// TwinCAT 3 PLC project PD30CTBxx
// Title: PD30CTBxx
// Company: iMusic AS
// Author: Jakob Bak
// ProjectVersion: 0.0.1.0
// Description: TwinCAT Library for PD30CTB* series Diffuse-reflective Photoelectric Sensors from Carlo Gavazzi
// ProgramVersion: 3.1.4024.0
// libraries:
//   Tc2_Standard, * (Beckhoff Automation GmbH)
//   Tc2_System, * (Beckhoff Automation GmbH)
//   Tc3_Module, * (Beckhoff Automation GmbH)
// project tree:
//   DUTs/ ST_PD30CTBxx.TcDUT
//   / PlcTask.TcTTO
//   POUs/ MAIN.TcPOU
//   Version/ Global_Version.TcGVL
// real-time tasks:
//   TASK PlcTask: cycle T#10ms, priority 20, ADS port 350

CONFIGURATION PD30CTBxx
    RESOURCE PLC ON TwinCAT3
        TASK PlcTask(INTERVAL := T#10ms, PRIORITY := 20);
        PROGRAM MAIN WITH PlcTask : MAIN;
    END_RESOURCE
END_CONFIGURATION

// ---- DUTs/ST_PD30CTBxx.TcDUT

TYPE ST_PD30CTBxx :
STRUCT
	bAnalogueValue				AT%I* : UINT;
	bSwitchingSignalChannel_1	AT%I* : BIT;
	bSwitchingSignalChannel_2	AT%I* : BIT;
	bDustAlarm_1				AT%I* : BIT;
	bDustAlarm_2				AT%I* : BIT;
	bTemperatureAlarm			AT%I* : BIT;
	bShortCircuit				AT%I* : BIT;
	bSwitchingOutput_1			AT%I* : BIT;
	bSwitchingOutput_2			AT%I* : BIT;
	bApplicationFunctionOutput	AT%I* : BIT;
END_STRUCT
END_TYPE

// ---- Version/Global_Version.TcGVL
{attribute 'TcGenerated'}
{attribute 'no-analysis'}
{attribute 'linkalways'}
// This function has been automatically generated from the project information.
VAR_GLOBAL CONSTANT
	{attribute 'const_non_replaced'}
	stLibVersion_PD30CTBxx : ST_LibVersion := (iMajor := 0, iMinor := 0, iBuild := 1, iRevision := 0, nFlags := 1, sVersion := '0.0.1.0');
END_VAR

// ---- POUs/MAIN.TcPOU
PROGRAM MAIN
VAR
END_VAR

END_PROGRAM
